(* PLC project paper-machine, Generated TextualNotationConverter 1.0 *)
(* stored: creationDateTime 2025-07-30T12:00:00, modificationDateTime 2025-01-30T12:00:00 *)

FUNCTION_BLOCK ANALOG_IN
  VAR_INPUT
    Name : STRING;
    Description : STRING;
    Raw_Signal : REAL;
    PV_High : REAL;
    PV_Low : REAL;
    Scaling_Slope : REAL;
    Scaling_Offset : REAL;
    Alarm_Enable : BOOL;
  END_VAR
  VAR_OUTPUT
    PV : REAL;
    High_Alarm : BOOL;
    Low_Alarm : BOOL;
    General_Fault : BOOL;
  END_VAR

            
          
END_FUNCTION_BLOCK

FUNCTION_BLOCK MOTOR_VSD
  VAR_INPUT
    Name : STRING;
    Description : STRING;
    Start_Cmd : BOOL;
    Stop_Cmd : BOOL;
    Speed_SP : REAL;
    Accel_Ramp : STRING;
    Decel_Ramp : STRING;
    Inhibit : BOOL;
  END_VAR
  VAR_OUTPUT
    Speed_Out : REAL;
    FB_Running : BOOL;
    FB_Fault : BOOL;
    FB_Ready : BOOL;
    FB_ActualSpeed : REAL;
    Alarm_Speed_Deviation : BOOL;
    Alarm_Comm_Fail : BOOL;
  END_VAR

            
          
END_FUNCTION_BLOCK

FUNCTION_BLOCK PID_BASIC
  VAR_INPUT
    Name : STRING;
    Description : STRING;
    AUTO : BOOL;
    PV : REAL;
    SP : REAL;
    MV_MIN : REAL;
    MV_MAX : REAL;
    X0 : REAL;
    KP : REAL;
    TR : REAL;
    TD : REAL;
    PV_High : REAL;
    PV_Low : REAL;
    Deviation_Limit : REAL;
    Inhibit : BOOL;
  END_VAR
  VAR_OUTPUT
    PV_High_Alarm : BOOL;
    PV_Low_Alarm : BOOL;
    Deviation_Alarm : BOOL;
    XOUT : REAL;
  END_VAR

            
          
END_FUNCTION_BLOCK

FUNCTION_BLOCK VALVE_ELECTRIC
  VAR_INPUT
    Name : STRING;
    Description : STRING;
    Control_Signal : REAL;
    Manual_Mode : BOOL;
    Manual_Position : REAL;
    Open_Limit : REAL;
    Close_Limit : REAL;
    Timeout : STRING;
    Inhibit : BOOL;
  END_VAR
  VAR_OUTPUT
    Valve_Position : REAL;
    Feedback_Pos : REAL;
    Valve_Moving : BOOL;
    Position_Error : BOOL;
    Alarm : BOOL;
  END_VAR

            
          
END_FUNCTION_BLOCK

FUNCTION_BLOCK VALVE_ON_OFF
  VAR_INPUT
    Name : STRING;
    Description : STRING;
    Open_Cmd : BOOL;
    Close_Cmd : BOOL;
    Timeout : STRING;
    Inhibit : BOOL;
  END_VAR
  VAR_OUTPUT
    FB_Opened : BOOL;
    FB_Closed : BOOL;
    Valve_Open_Out : BOOL;
    Valve_Close_Out : BOOL;
    Alarm_Position_Error : BOOL;
    Alarm_General : BOOL;
  END_VAR

            
          
END_FUNCTION_BLOCK

PROGRAM Section2
  VAR
    LT_101_Flow_PV : REAL;
    FC_101_MV_to_FV106 : REAL;
    M_102_VSD_Speed_Out : REAL;
    Flow_Deviation_Alarm_30s : BOOL;
    Flow_High_Alarm : BOOL;
    Flow_Low_Alarm : BOOL;
    M_102_Start_Request : BOOL;
    M_102_Stop_Request : BOOL;
  END_VAR
  VAR
    LT-101 : ANALOG_IN;
    FC-101 : PID_BASIC;
    M-102 : MOTOR_VSD;
    FV-106 : VALVE_ELECTRIC;
    LV-103 : VALVE_ELECTRIC;
    XV-102 : VALVE_ON_OFF;
    XV-104 : VALVE_ON_OFF;
    XV-105 : VALVE_ON_OFF;
  END_VAR
  VAR  (* added by the conversion: wires and edge detectors of the diagram *)
    _OR5_OUT : BOOL;
  END_VAR

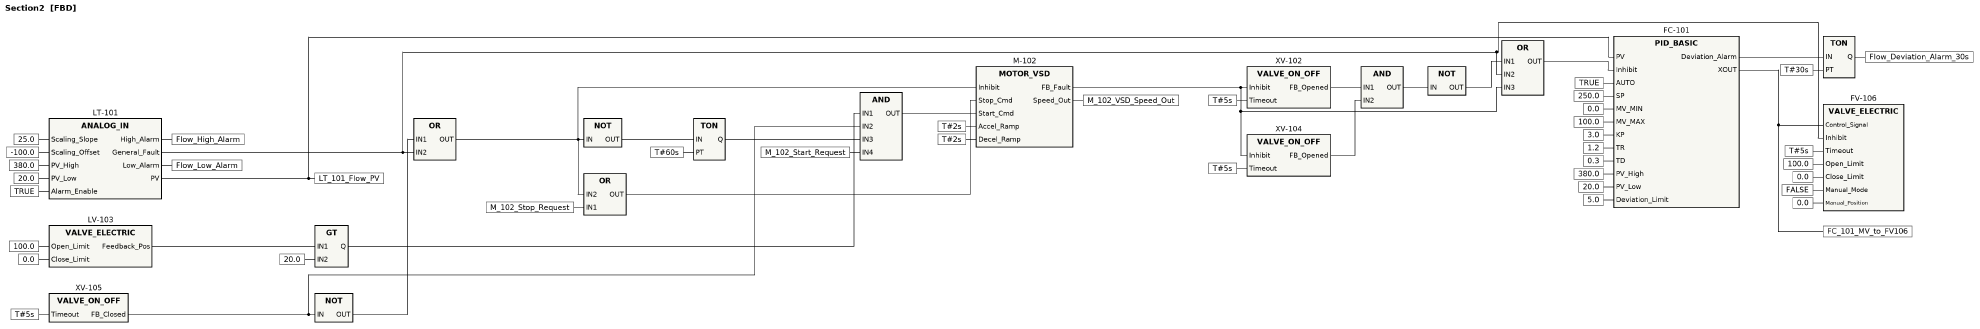
(* FBD diagram, written out as Structured Text *)
LT-101(Scaling_Slope := 25.0, Scaling_Offset := -100.0, PV_High := 380.0, PV_Low := 20.0, Alarm_Enable := TRUE);
XV-105(Timeout := T#5s);
_OR5_OUT := NOT XV-105.FB_Closed OR LT-101.General_Fault;
LV-103(Open_Limit := 100.0, Close_Limit := 0.0);
M-102(Inhibit := _OR5_OUT, Stop_Cmd := _OR5_OUT OR M_102_Stop_Request, Start_Cmd := LV-103.Feedback_Pos > 20.0 AND XV-105.FB_Closed AND TON(NOT _OR5_OUT, T#60s) AND M_102_Start_Request, Accel_Ramp := T#2s, Decel_Ramp := T#2s);
XV-102(Inhibit := M-102.FB_Fault, Timeout := T#5s);
XV-104(Inhibit := M-102.FB_Fault, Timeout := T#5s);
FC-101(PV := LT-101.PV, Inhibit := NOT (XV-102.FB_Opened AND XV-104.FB_Opened) OR LT-101.General_Fault OR M-102.FB_Fault, AUTO := TRUE, SP := 250.0, MV_MIN := 0.0, MV_MAX := 100.0, KP := 3.0, TR := 1.2, TD := 0.3, PV_High := 380.0, PV_Low := 20.0, Deviation_Limit := 5.0);
FC_101_MV_to_FV106 := FC-101.XOUT;
Flow_Deviation_Alarm_30s := TON(FC-101.Deviation_Alarm, T#30s);
Flow_High_Alarm := LT-101.High_Alarm;
Flow_Low_Alarm := LT-101.Low_Alarm;
LT_101_Flow_PV := LT-101.PV;
M_102_VSD_Speed_Out := M-102.Speed_Out;
FV-106(Control_Signal := FC-101.XOUT, Inhibit := LT-101.General_Fault, Timeout := T#5s, Open_Limit := 100.0, Close_Limit := 0.0, Manual_Mode := FALSE, Manual_Position := 0.0);
END_PROGRAM

FUNCTION_BLOCK BOOL_IN
  VAR_INPUT
    Name : STRING;
    Description : STRING;
    Bool_In : BOOL;
    Alarm_OnTrue : BOOL;
    Alarm_OnFalse : BOOL;
    Latch_Enable : BOOL;
    Reset_Latch : BOOL;
  END_VAR
  VAR_OUTPUT
    Bool_Out : BOOL;
    Alarm_Active : BOOL;
    Latched_Status : BOOL;
  END_VAR

            
          
END_FUNCTION_BLOCK

FUNCTION_BLOCK DIGITAL_IN
  VAR_INPUT
    Name : STRING;
    Description : STRING;
    DI_Raw : BOOL;
    DebounceTime : STRING;
    EnableAlarm : BOOL;
  END_VAR
  VAR_OUTPUT
    DI_Out : BOOL;
    Fault_State : BOOL;
  END_VAR

            
          
END_FUNCTION_BLOCK

FUNCTION_BLOCK DUTY_STANDBY
  VAR_INPUT
    Name : STRING;
    Description : STRING;
    Enable : BOOL;
    StartRequest : BOOL;
    AlternateEnable : BOOL;
    ForcePumpA : BOOL;
    ForcePumpB : BOOL;
    DutyElapsed : BOOL;
    MinRunElapsed : BOOL;
    SwitchoverDelayElapsed : BOOL;
    StartTimeoutElapsed : BOOL;
    PumpA_RunFB : BOOL;
    PumpB_RunFB : BOOL;
    PumpA_Fault : BOOL;
    PumpB_Fault : BOOL;
    Reset : BOOL;
    Inhibit : BOOL;
  END_VAR
  VAR_OUTPUT
    CmdPumpA : BOOL;
    CmdPumpB : BOOL;
    ActiveIsA : BOOL;
    SwitchedDueToDuty : BOOL;
    SwitchedDueToFailure : BOOL;
    Alarm_FailedStart_A : BOOL;
    Alarm_FailedStart_B : BOOL;
    Alarm_NoAvailablePump : BOOL;
  END_VAR

            
          
END_FUNCTION_BLOCK

FUNCTION_BLOCK MOTOR_2SPD
  VAR_INPUT
    Name : STRING;
    Description : STRING;
    Start_Cmd : BOOL;
    Stop_Cmd : BOOL;
    Speed_High_Cmd : BOOL;
    Speed_Low_Cmd : BOOL;
    Inhibit : BOOL;
  END_VAR
  VAR_OUTPUT
    Motor_Start_Out : BOOL;
    FB_Running : BOOL;
    FB_Trip : BOOL;
    FB_HighSpeed : BOOL;
    FB_LowSpeed : BOOL;
    Alarm_Speed_Error : BOOL;
  END_VAR

            
          
END_FUNCTION_BLOCK

FUNCTION_BLOCK MOTOR_ON_OFF
  VAR_INPUT
    Name : STRING;
    Description : STRING;
    Start_Cmd : BOOL;
    Stop_Cmd : BOOL;
    Start_Delay : STRING;
    MinRunTime : STRING;
    Inhibit : BOOL;
  END_VAR
  VAR_OUTPUT
    Motor_Start_Out : BOOL;
    FB_Running : BOOL;
    FB_Trip : BOOL;
    Alarm_Start_Fail : BOOL;
    Alarm_Stop_Fail : BOOL;
  END_VAR

            
          
END_FUNCTION_BLOCK

FUNCTION_BLOCK RATIO_CONTROL
  VAR_INPUT
    Name : STRING;
    Description : STRING;
    Auto : BOOL;
    PrimaryPV : REAL;
    SecondaryPV : REAL;
    RatioSP : REAL;
    Bias : REAL;
    TrimKp : REAL;
    TrimTi : STRING;
    MV_MIN : REAL;
    MV_MAX : REAL;
    ManOut : REAL;
    Inhibit : BOOL;
  END_VAR
  VAR_OUTPUT
    SlaveSP : REAL;
    ActiveRatio : REAL;
    RatioErr : REAL;
  END_VAR

            
          
END_FUNCTION_BLOCK

FUNCTION_BLOCK SPLIT_RANGE
  VAR_INPUT
    Name : STRING;
    Description : STRING;
    IN : REAL;
    Split_Point : REAL;
    Output1_Start : REAL;
    Output1_End : REAL;
    Output2_Start : REAL;
    Output2_End : REAL;
  END_VAR
  VAR_OUTPUT
    OUT1 : REAL;
    OUT2 : REAL;
  END_VAR

            
          
END_FUNCTION_BLOCK

FUNCTION_BLOCK VOTING_ANALOG
  VAR_INPUT
    Name : STRING;
    Description : STRING;
    Input1 : REAL;
    Input2 : REAL;
    Input3 : REAL;
    Deviation_Limit : REAL;
    Voting_Scheme : STRING;
    EnableAlarm : BOOL;
    Inhibit : BOOL;
  END_VAR
  VAR_OUTPUT
    Voted_Output : REAL;
    Sensor1_Fault : BOOL;
    Sensor2_Fault : BOOL;
    Sensor3_Fault : BOOL;
    Alarm_Voting_Error : BOOL;
    Healthy_Sensors_Count : INT;
  END_VAR

            
          
END_FUNCTION_BLOCK

PROGRAM Section3
  VAR
    TT_103_Temperature_PV : REAL;
    PT_101_Pressure_PV : REAL;
    TIC_104_RSP_to_FC_203 : REAL;
    PIC_101_RSP_to_FC_202 : REAL;
    FC_203_MV_to_SV_203 : REAL;
    FC_202_MV_to_FV_202 : REAL;
  END_VAR
  VAR
    TT-103 : ANALOG_IN;
    PT-101 : ANALOG_IN;
    TIC-104 : PID_BASIC;
    PIC-101 : PID_BASIC;
    FC-203 : PID_BASIC;
    FC-202 : PID_BASIC;
    SV-203 : VALVE_ELECTRIC;
    FV-202 : VALVE_ELECTRIC;
  END_VAR
  VAR  (* added by the conversion: wires and edge detectors of the diagram *)
    _OR59_OUT : BOOL;
  END_VAR

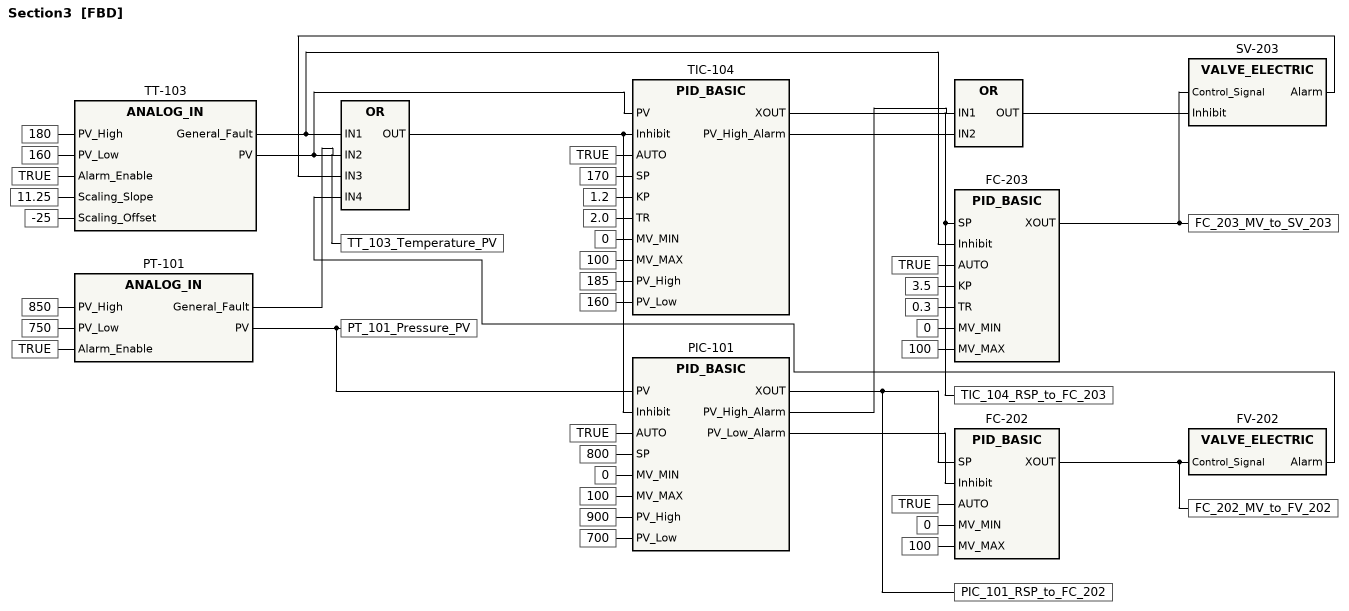
(* FBD diagram, written out as Structured Text *)
PT-101(PV_High := 850, PV_Low := 750, Alarm_Enable := TRUE);
TT-103(PV_High := 180, PV_Low := 160, Alarm_Enable := TRUE, Scaling_Slope := 11.25, Scaling_Offset := -25);
TIC-104(PV := TT-103.PV, Inhibit := _OR59_OUT, AUTO := TRUE, SP := 170, KP := 1.2, TR := 2.0, MV_MIN := 0, MV_MAX := 100, PV_High := 185, PV_Low := 160);
FC-203(SP := TIC-104.XOUT, Inhibit := TT-103.General_Fault, AUTO := TRUE, KP := 3.5, TR := 0.3, MV_MIN := 0, MV_MAX := 100);
SV-203(Control_Signal := FC-203.XOUT, Inhibit := PIC-101.PV_High_Alarm OR TIC-104.PV_High_Alarm);
FV-202(Control_Signal := FC-202.XOUT);
_OR59_OUT := TT-103.General_Fault OR PT-101.General_Fault OR SV-203.Alarm OR FV-202.Alarm;
PIC-101(PV := PT-101.PV, Inhibit := _OR59_OUT, AUTO := TRUE, SP := 800, MV_MIN := 0, MV_MAX := 100, PV_High := 900, PV_Low := 700);
FC-202(SP := PIC-101.XOUT, Inhibit := PIC-101.PV_Low_Alarm, AUTO := TRUE, MV_MIN := 0, MV_MAX := 100);
FC_202_MV_to_FV_202 := FC-202.XOUT;
FC_203_MV_to_SV_203 := FC-203.XOUT;
PIC_101_RSP_to_FC_202 := PIC-101.XOUT;
PT_101_Pressure_PV := PT-101.PV;
TIC_104_RSP_to_FC_203 := TIC-104.XOUT;
TT_103_Temperature_PV := TT-103.PV;
END_PROGRAM

PROGRAM Section4
  VAR
    PIT103_Pressure_kPa : REAL;
    PT101_UpstreamPressure_kPa : REAL;
    DT301_PulpDensity_Pct : REAL;
    PIC104_ControlOutput_to_FV106_Pct : REAL;
    FV106_ValvePositionFeedback_Pct : REAL;
  END_VAR
  VAR
    DT-301 : ANALOG_IN;
    PIT-103 : ANALOG_IN;
    PT-101 : ANALOG_IN;
    PIC-104 : PID_BASIC;
    FV-106 : VALVE_ELECTRIC;
    XV-102 : VALVE_ON_OFF;
    XV-107 : VALVE_ON_OFF;
    XV-102-OPEN-FB : DIGITAL_IN;
    XV-107-OPEN-FB : DIGITAL_IN;
    PERM-XV102-OPEN : BOOL_IN;
    PERM-XV107-OPEN : BOOL_IN;
  END_VAR
  VAR  (* added by the conversion: wires and edge detectors of the diagram *)
    _OR104_OUT : BOOL;
    _OR106_OUT : BOOL;
    _NOT109_OUT : BOOL;
  END_VAR

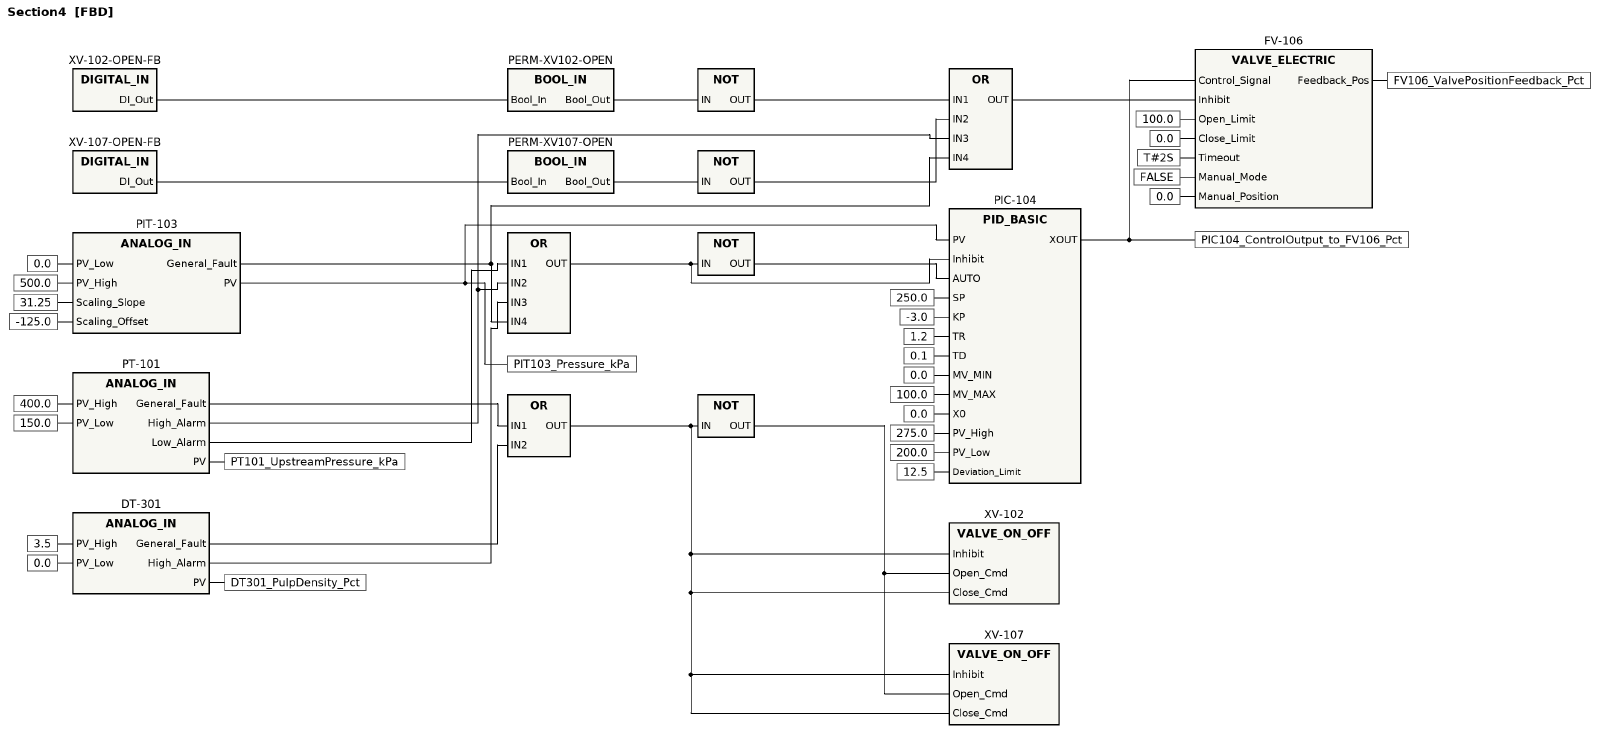
(* FBD diagram, written out as Structured Text *)
DT-301(PV_High := 3.5, PV_Low := 0.0);
DT301_PulpDensity_Pct := DT-301.PV;
PIT-103(PV_Low := 0.0, PV_High := 500.0, Scaling_Slope := 31.25, Scaling_Offset := -125.0);
PT-101(PV_High := 400.0, PV_Low := 150.0);
_OR104_OUT := PT-101.Low_Alarm OR PT-101.High_Alarm OR DT-301.High_Alarm OR PIT-103.General_Fault;
PIC-104(PV := PIT-103.PV, Inhibit := _OR104_OUT, AUTO := NOT _OR104_OUT, SP := 250.0, KP := -3.0, TR := 1.2, TD := 0.1, MV_MIN := 0.0, MV_MAX := 100.0, X0 := 0.0, PV_High := 275.0, PV_Low := 200.0, Deviation_Limit := 12.5);
XV-102-OPEN-FB();
PERM-XV102-OPEN(Bool_In := XV-102-OPEN-FB.DI_Out);
XV-107-OPEN-FB();
PERM-XV107-OPEN(Bool_In := XV-107-OPEN-FB.DI_Out);
FV-106(Control_Signal := PIC-104.XOUT, Inhibit := NOT PERM-XV102-OPEN.Bool_Out OR NOT PERM-XV107-OPEN.Bool_Out OR PT-101.High_Alarm OR PIT-103.General_Fault, Open_Limit := 100.0, Close_Limit := 0.0, Timeout := T#2S, Manual_Mode := FALSE, Manual_Position := 0.0);
FV106_ValvePositionFeedback_Pct := FV-106.Feedback_Pos;
PIC104_ControlOutput_to_FV106_Pct := PIC-104.XOUT;
PIT103_Pressure_kPa := PIT-103.PV;
PT101_UpstreamPressure_kPa := PT-101.PV;
_OR106_OUT := PT-101.General_Fault OR DT-301.General_Fault;
_NOT109_OUT := NOT _OR106_OUT;
XV-102(Inhibit := _OR106_OUT, Open_Cmd := _NOT109_OUT, Close_Cmd := _OR106_OUT);
XV-107(Inhibit := _OR106_OUT, Open_Cmd := _NOT109_OUT, Close_Cmd := _OR106_OUT);
END_PROGRAM

PROGRAM Section5
  VAR
    AT102_pH_PV : REAL;
    AT107_pH_PV : REAL;
    TIT106_Temperature_PV : REAL;
    LIC102_MV_to_FV101 : REAL;
    TIC106_MV_to_FV103 : REAL;
    LIC104_MV_to_XV104 : REAL;
  END_VAR
  VAR
    AT-102 : ANALOG_IN;
    AT-107 : ANALOG_IN;
    TIT-106 : ANALOG_IN;
    LIC-102 : PID_BASIC;
    TIC-106 : PID_BASIC;
    LIC-104 : PID_BASIC;
    FV-101 : VALVE_ELECTRIC;
    FV-103 : VALVE_ELECTRIC;
    XV-104 : VALVE_ELECTRIC;
  END_VAR

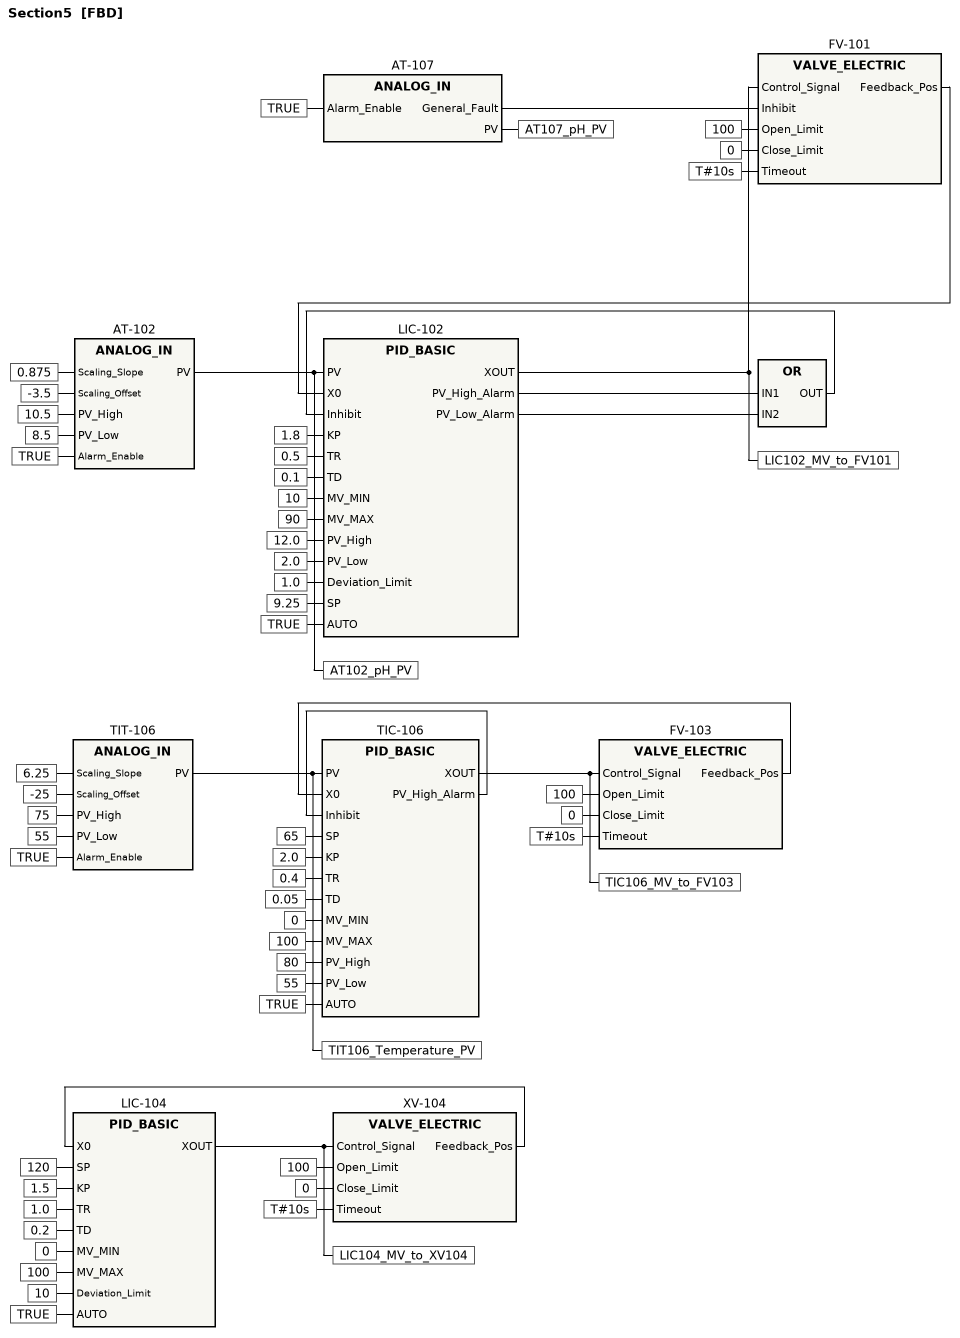
(* FBD diagram, written out as Structured Text *)
AT-102(Scaling_Slope := 0.875, Scaling_Offset := -3.5, PV_High := 10.5, PV_Low := 8.5, Alarm_Enable := TRUE);
AT102_pH_PV := AT-102.PV;
AT-107(Alarm_Enable := TRUE);
AT107_pH_PV := AT-107.PV;
FV-101(Control_Signal := LIC-102.XOUT, Inhibit := AT-107.General_Fault, Open_Limit := 100, Close_Limit := 0, Timeout := T#10s);
LIC-102(PV := AT-102.PV, X0 := FV-101.Feedback_Pos, Inhibit := LIC-102.PV_High_Alarm OR LIC-102.PV_Low_Alarm, KP := 1.8, TR := 0.5, TD := 0.1, MV_MIN := 10, MV_MAX := 90, PV_High := 12.0, PV_Low := 2.0, Deviation_Limit := 1.0, SP := 9.25, AUTO := TRUE);
LIC102_MV_to_FV101 := LIC-102.XOUT;
XV-104(Control_Signal := LIC-104.XOUT, Open_Limit := 100, Close_Limit := 0, Timeout := T#10s);
LIC-104(X0 := XV-104.Feedback_Pos, SP := 120, KP := 1.5, TR := 1.0, TD := 0.2, MV_MIN := 0, MV_MAX := 100, Deviation_Limit := 10, AUTO := TRUE);
LIC104_MV_to_XV104 := LIC-104.XOUT;
TIT-106(Scaling_Slope := 6.25, Scaling_Offset := -25, PV_High := 75, PV_Low := 55, Alarm_Enable := TRUE);
FV-103(Control_Signal := TIC-106.XOUT, Open_Limit := 100, Close_Limit := 0, Timeout := T#10s);
TIC-106(PV := TIT-106.PV, X0 := FV-103.Feedback_Pos, Inhibit := TIC-106.PV_High_Alarm, SP := 65, KP := 2.0, TR := 0.4, TD := 0.05, MV_MIN := 0, MV_MAX := 100, PV_High := 80, PV_Low := 55, AUTO := TRUE);
TIC106_MV_to_FV103 := TIC-106.XOUT;
TIT106_Temperature_PV := TIT-106.PV;
END_PROGRAM

PROGRAM Section6
  VAR
    CT501_Consistency_PV_Pct : REAL;
    FC502_MV_to_FV502_Pct : REAL;
    SELT501_SEL_PV_WsPerMm2 : REAL;
    SELC501_MV_to_PGA501_Pct : REAL;
    LT501_Level_PV_Pct : REAL;
    PT502_Pressure_PV_kPa : REAL;
    PGT501_PlateGap_PV_mm : REAL;
  END_VAR
  VAR
    CT-501 : ANALOG_IN;
    FC-502 : PID_BASIC;
    FV-502 : VALVE_ELECTRIC;
    LT-501 : ANALOG_IN;
    M-501 : MOTOR_ON_OFF;
    PT-502 : ANALOG_IN;
    SELC-501 : PID_BASIC;
    PGT-501 : ANALOG_IN;
    PGA-501 : VALVE_ELECTRIC;
    SELT-501 : ANALOG_IN;
    INTLK-M501-RUNNING : BOOL_IN;
    INTLK-PLATE-GAP-IN-RANGE : BOOL_IN;
    INTLK-LEVEL-ABOVE-20 : BOOL_IN;
    PERM-PT502-IN-RANGE : BOOL_IN;
  END_VAR
  VAR  (* added by the conversion: wires and edge detectors of the diagram *)
    _OR217_OUT : BOOL;
    _OR219_OUT : BOOL;
    _OR221_OUT : BOOL;
    _OR213_OUT : BOOL;
  END_VAR

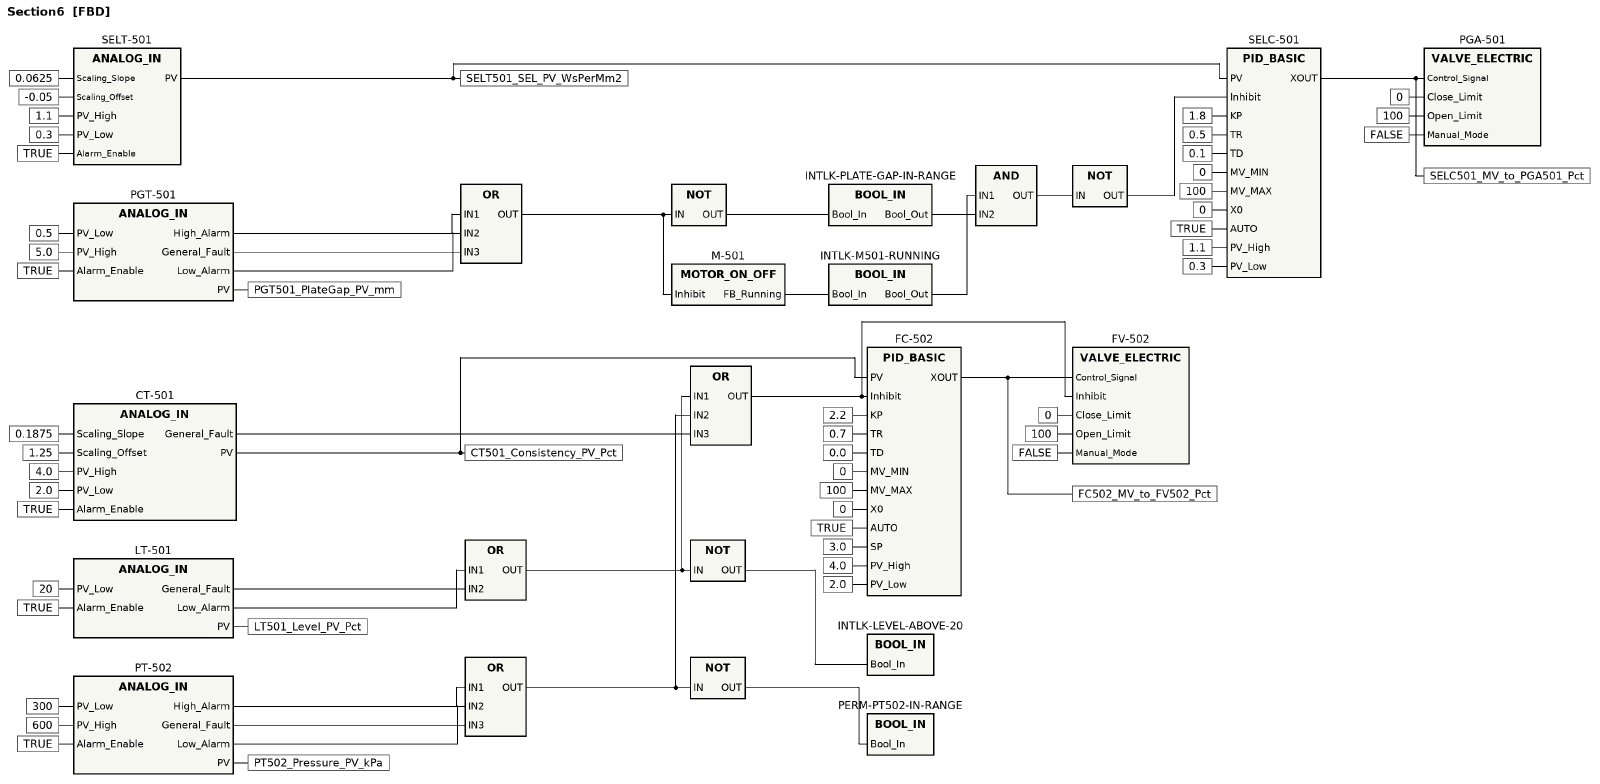
(* FBD diagram, written out as Structured Text *)
CT-501(Scaling_Slope := 0.1875, Scaling_Offset := 1.25, PV_High := 4.0, PV_Low := 2.0, Alarm_Enable := TRUE);
CT501_Consistency_PV_Pct := CT-501.PV;
LT-501(PV_Low := 20, Alarm_Enable := TRUE);
_OR217_OUT := LT-501.Low_Alarm OR LT-501.General_Fault;
PT-502(PV_Low := 300, PV_High := 600, Alarm_Enable := TRUE);
_OR219_OUT := PT-502.High_Alarm OR PT-502.Low_Alarm OR PT-502.General_Fault;
_OR221_OUT := _OR217_OUT OR _OR219_OUT OR CT-501.General_Fault;
FC-502(PV := CT-501.PV, Inhibit := _OR221_OUT, KP := 2.2, TR := 0.7, TD := 0.0, MV_MIN := 0, MV_MAX := 100, X0 := 0, AUTO := TRUE, SP := 3.0, PV_High := 4.0, PV_Low := 2.0);
FC502_MV_to_FV502_Pct := FC-502.XOUT;
LT501_Level_PV_Pct := LT-501.PV;
PGT-501(PV_Low := 0.5, PV_High := 5.0, Alarm_Enable := TRUE);
PGT501_PlateGap_PV_mm := PGT-501.PV;
PT502_Pressure_PV_kPa := PT-502.PV;
SELT-501(Scaling_Slope := 0.0625, Scaling_Offset := -0.05, PV_High := 1.1, PV_Low := 0.3, Alarm_Enable := TRUE);
_OR213_OUT := PGT-501.High_Alarm OR PGT-501.Low_Alarm OR PGT-501.General_Fault;
M-501(Inhibit := _OR213_OUT);
INTLK-M501-RUNNING(Bool_In := M-501.FB_Running);
INTLK-PLATE-GAP-IN-RANGE(Bool_In := NOT _OR213_OUT);
SELC-501(PV := SELT-501.PV, Inhibit := NOT (INTLK-M501-RUNNING.Bool_Out AND INTLK-PLATE-GAP-IN-RANGE.Bool_Out), KP := 1.8, TR := 0.5, TD := 0.1, MV_MIN := 0, MV_MAX := 100, X0 := 0, AUTO := TRUE, PV_High := 1.1, PV_Low := 0.3);
SELC501_MV_to_PGA501_Pct := SELC-501.XOUT;
SELT501_SEL_PV_WsPerMm2 := SELT-501.PV;
FV-502(Control_Signal := FC-502.XOUT, Inhibit := _OR221_OUT, Close_Limit := 0, Open_Limit := 100, Manual_Mode := FALSE);
PGA-501(Control_Signal := SELC-501.XOUT, Close_Limit := 0, Open_Limit := 100, Manual_Mode := FALSE);
INTLK-LEVEL-ABOVE-20(Bool_In := NOT _OR217_OUT);
PERM-PT502-IN-RANGE(Bool_In := NOT _OR219_OUT);
END_PROGRAM

PROGRAM Section7
  VAR
    CT_601_PV : REAL;
    FT_601_PV : REAL;
    FT_601_SP : REAL;
    PIT_601_PV : REAL;
    VT_601_PV : REAL;
    FS_601_MinFlow_OK : BOOL;
    P_601_Run_OK : BOOL;
    FFIC601_Bias : REAL;
    ALM_601 : BOOL;
    ALM_601_High : BOOL;
    ALM_601_Low : BOOL;
    ALM_602 : BOOL;
    ALM_603 : BOOL;
    ALM_604 : BOOL;
    Process_Permissives_OK : BOOL;
    MasterInhibit : BOOL;
    CT601_RateHigh : BOOL;
  END_VAR
  VAR
    CT-601 : ANALOG_IN;
    FT-601 : ANALOG_IN;
    PIT-601 : ANALOG_IN;
    VT-601 : ANALOG_IN;
    FS-601 : BOOL_IN;
    P-601_RUN : BOOL_IN;
    FV-601 : VALVE_ELECTRIC;
    FIC-601 : PID_BASIC;
    FFIC-601 : RATIO_CONTROL;
    ProcessUpset_Timer : TON;
  END_VAR
  VAR  (* added by the conversion: wires and edge detectors of the diagram *)
    _OR288_OUT : BOOL;
    _OR289_OUT : BOOL;
    _OR290_OUT : BOOL;
    _NOT291_OUT : BOOL;
  END_VAR

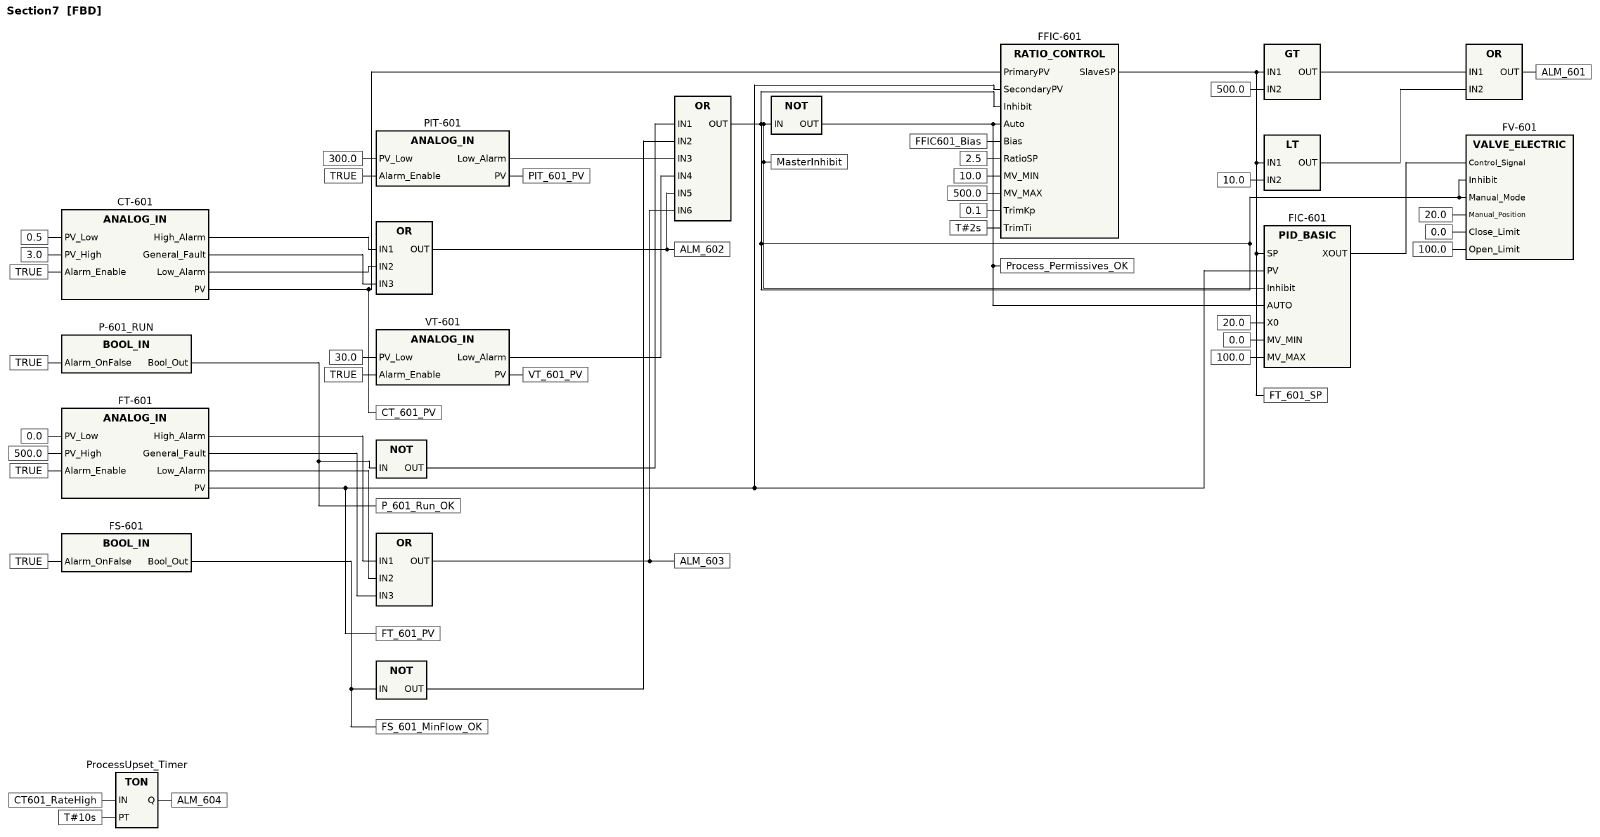
(* FBD diagram, written out as Structured Text *)
CT-601(PV_Low := 0.5, PV_High := 3.0, Alarm_Enable := TRUE);
FT-601(PV_Low := 0.0, PV_High := 500.0, Alarm_Enable := TRUE);
P-601_RUN(Alarm_OnFalse := TRUE);
FS-601(Alarm_OnFalse := TRUE);
PIT-601(PV_Low := 300.0, Alarm_Enable := TRUE);
VT-601(PV_Low := 30.0, Alarm_Enable := TRUE);
_OR288_OUT := CT-601.High_Alarm OR CT-601.Low_Alarm OR CT-601.General_Fault;
_OR289_OUT := FT-601.High_Alarm OR FT-601.Low_Alarm OR FT-601.General_Fault;
_OR290_OUT := NOT P-601_RUN.Bool_Out OR NOT FS-601.Bool_Out OR PIT-601.Low_Alarm OR VT-601.Low_Alarm OR _OR288_OUT OR _OR289_OUT;
_NOT291_OUT := NOT _OR290_OUT;
FFIC-601(PrimaryPV := CT-601.PV, SecondaryPV := FT-601.PV, Inhibit := _OR290_OUT, Auto := _NOT291_OUT, Bias := FFIC601_Bias, RatioSP := 2.5, MV_MIN := 10.0, MV_MAX := 500.0, TrimKp := 0.1, TrimTi := T#2s);
ALM_601 := FFIC-601.SlaveSP > 500.0 OR FFIC-601.SlaveSP < 10.0;
ALM_602 := _OR288_OUT;
ALM_603 := _OR289_OUT;
ProcessUpset_Timer(IN := CT601_RateHigh, PT := T#10s);
ALM_604 := ProcessUpset_Timer.Q;
CT_601_PV := CT-601.PV;
FS_601_MinFlow_OK := FS-601.Bool_Out;
FT_601_PV := FT-601.PV;
FT_601_SP := FFIC-601.SlaveSP;
MasterInhibit := _OR290_OUT;
PIT_601_PV := PIT-601.PV;
P_601_Run_OK := P-601_RUN.Bool_Out;
Process_Permissives_OK := _NOT291_OUT;
VT_601_PV := VT-601.PV;
FIC-601(SP := FFIC-601.SlaveSP, PV := FT-601.PV, Inhibit := _OR290_OUT, AUTO := _NOT291_OUT, X0 := 20.0, MV_MIN := 0.0, MV_MAX := 100.0);
FV-601(Control_Signal := FIC-601.XOUT, Inhibit := _OR290_OUT, Manual_Mode := _OR290_OUT, Manual_Position := 20.0, Close_Limit := 0.0, Open_Limit := 100.0);
END_PROGRAM

PROGRAM Section8
  VAR
    MM701_Raw_mA : REAL;
    PT701_Raw : REAL;
    TT102_Raw : REAL;
    HS701_ON : BOOL;
    CS701_ON : BOOL;
    SB701_SheetBreak : BOOL;
    MM701_Moisture_PV : REAL;
    PT701_HydraulicPressure_PV : REAL;
    TT102_ShowerWaterTemp_PV : REAL;
    PV101_Pressure_Command_Pct : REAL;
    PV101_Position_Feedback_Pct : REAL;
    ESD_Trip : BOOL;
  END_VAR
  VAR
    MM-701 : ANALOG_IN;
    PT-701 : ANALOG_IN;
    TT-102 : ANALOG_IN;
    LIC-701 : PID_BASIC;
    PV-101 : VALVE_ELECTRIC;
    HS-701 : BOOL_IN;
    CS-701 : BOOL_IN;
    SB-701 : BOOL_IN;
  END_VAR
  VAR  (* added by the conversion: wires and edge detectors of the diagram *)
    _OR348_OUT : BOOL;
  END_VAR

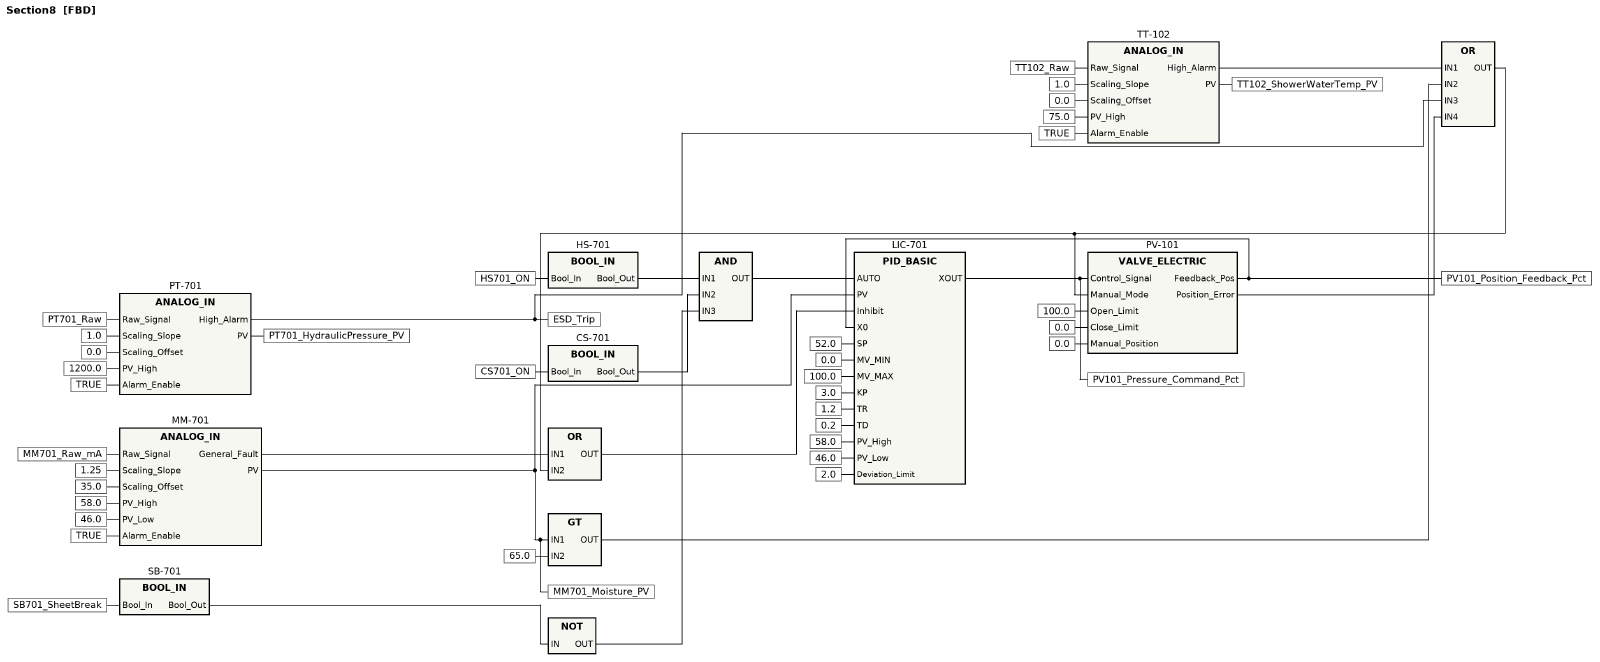
(* FBD diagram, written out as Structured Text *)
PT-701(Raw_Signal := PT701_Raw, Scaling_Slope := 1.0, Scaling_Offset := 0.0, PV_High := 1200.0, Alarm_Enable := TRUE);
ESD_Trip := PT-701.High_Alarm;
MM-701(Raw_Signal := MM701_Raw_mA, Scaling_Slope := 1.25, Scaling_Offset := 35.0, PV_High := 58.0, PV_Low := 46.0, Alarm_Enable := TRUE);
MM701_Moisture_PV := MM-701.PV;
PT701_HydraulicPressure_PV := PT-701.PV;
HS-701(Bool_In := HS701_ON);
CS-701(Bool_In := CS701_ON);
SB-701(Bool_In := SB701_SheetBreak);
TT-102(Raw_Signal := TT102_Raw, Scaling_Slope := 1.0, Scaling_Offset := 0.0, PV_High := 75.0, Alarm_Enable := TRUE);
_OR348_OUT := TT-102.High_Alarm OR MM-701.PV > 65.0 OR PT-701.High_Alarm OR PV-101.Position_Error;
LIC-701(AUTO := HS-701.Bool_Out AND CS-701.Bool_Out AND NOT SB-701.Bool_Out, PV := MM-701.PV, Inhibit := MM-701.General_Fault OR _OR348_OUT, X0 := PV-101.Feedback_Pos, SP := 52.0, MV_MIN := 0.0, MV_MAX := 100.0, KP := 3.0, TR := 1.2, TD := 0.2, PV_High := 58.0, PV_Low := 46.0, Deviation_Limit := 2.0);
PV-101(Control_Signal := LIC-701.XOUT, Manual_Mode := _OR348_OUT, Open_Limit := 100.0, Close_Limit := 0.0, Manual_Position := 0.0);
PV101_Position_Feedback_Pct := PV-101.Feedback_Pos;
PV101_Pressure_Command_Pct := LIC-701.XOUT;
TT102_ShowerWaterTemp_PV := TT-102.PV;
END_PROGRAM

PROGRAM Section9
  VAR
    F801_ExhaustFan_Speed_CMD_PCT : REAL;
    FV801_SteamFlowValve_Position_CMD_PCT : REAL;
    XV802_HotAirDamper_Position_CMD_PCT : REAL;
    WT801_DownstreamDriveRoll_Torque_CMD_PCT : REAL;
    XV802_Open_FB : BOOL;
    IR801_Available : BOOL;
  END_VAR
  VAR
    TT-801 : ANALOG_IN;
    TT-802 : ANALOG_IN;
    PT-801 : ANALOG_IN;
    IR-801 : ANALOG_IN;
    WT-801 : ANALOG_IN;
    F-801 : MOTOR_VSD;
    M-801 : MOTOR_ON_OFF;
    FV-801 : VALVE_ELECTRIC;
    XV-802 : VALVE_ELECTRIC;
    SC-801 : PID_BASIC;
    TC-801 : PID_BASIC;
    F-801_CTRL : PID_BASIC;
    WT-801_CTRL : PID_BASIC;
  END_VAR
  VAR  (* added by the conversion: wires and edge detectors of the diagram *)
    _OR401_OUT : BOOL;
    _OR397_OUT : BOOL;
  END_VAR

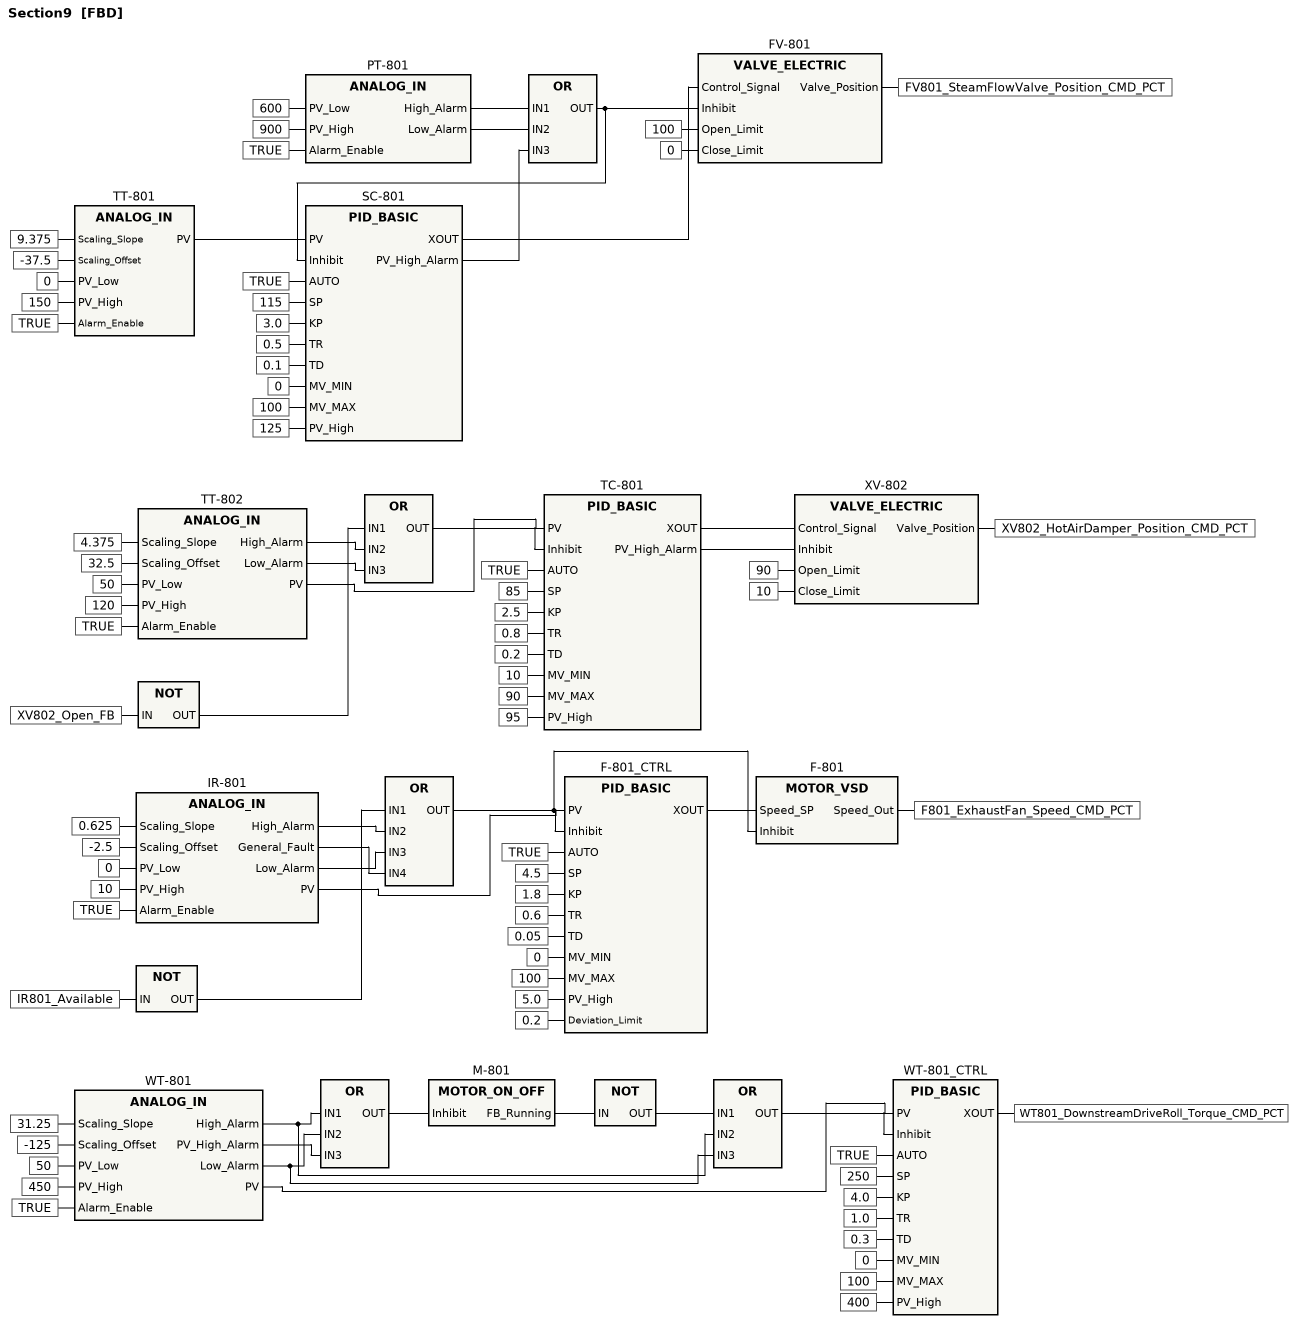
(* FBD diagram, written out as Structured Text *)
IR-801(Scaling_Slope := 0.625, Scaling_Offset := -2.5, PV_Low := 0, PV_High := 10, Alarm_Enable := TRUE);
_OR401_OUT := NOT IR801_Available OR IR-801.High_Alarm OR IR-801.Low_Alarm OR IR-801.General_Fault;
F-801_CTRL(PV := IR-801.PV, Inhibit := _OR401_OUT, AUTO := TRUE, SP := 4.5, KP := 1.8, TR := 0.6, TD := 0.05, MV_MIN := 0, MV_MAX := 100, PV_High := 5.0, Deviation_Limit := 0.2);
F-801(Speed_SP := F-801_CTRL.XOUT, Inhibit := _OR401_OUT);
F801_ExhaustFan_Speed_CMD_PCT := F-801.Speed_Out;
TT-801(Scaling_Slope := 9.375, Scaling_Offset := -37.5, PV_Low := 0, PV_High := 150, Alarm_Enable := TRUE);
PT-801(PV_Low := 600, PV_High := 900, Alarm_Enable := TRUE);
_OR397_OUT := PT-801.High_Alarm OR PT-801.Low_Alarm OR SC-801.PV_High_Alarm;
SC-801(PV := TT-801.PV, Inhibit := _OR397_OUT, AUTO := TRUE, SP := 115, KP := 3.0, TR := 0.5, TD := 0.1, MV_MIN := 0, MV_MAX := 100, PV_High := 125);
FV-801(Control_Signal := SC-801.XOUT, Inhibit := _OR397_OUT, Open_Limit := 100, Close_Limit := 0);
FV801_SteamFlowValve_Position_CMD_PCT := FV-801.Valve_Position;
WT-801(Scaling_Slope := 31.25, Scaling_Offset := -125, PV_Low := 50, PV_High := 450, Alarm_Enable := TRUE);
M-801(Inhibit := WT-801.High_Alarm OR WT-801.Low_Alarm OR WT-801.PV_High_Alarm);
WT-801_CTRL(PV := WT-801.PV, Inhibit := NOT M-801.FB_Running OR WT-801.High_Alarm OR WT-801.Low_Alarm, AUTO := TRUE, SP := 250, KP := 4.0, TR := 1.0, TD := 0.3, MV_MIN := 0, MV_MAX := 100, PV_High := 400);
WT801_DownstreamDriveRoll_Torque_CMD_PCT := WT-801_CTRL.XOUT;
TT-802(Scaling_Slope := 4.375, Scaling_Offset := 32.5, PV_Low := 50, PV_High := 120, Alarm_Enable := TRUE);
TC-801(PV := TT-802.PV, Inhibit := NOT XV802_Open_FB OR TT-802.High_Alarm OR TT-802.Low_Alarm, AUTO := TRUE, SP := 85, KP := 2.5, TR := 0.8, TD := 0.2, MV_MIN := 10, MV_MAX := 90, PV_High := 95);
XV-802(Control_Signal := TC-801.XOUT, Inhibit := TC-801.PV_High_Alarm, Open_Limit := 90, Close_Limit := 10);
XV802_HotAirDamper_Position_CMD_PCT := XV-802.Valve_Position;
END_PROGRAM

PROGRAM Section10
  VAR
    FT901_NipLoad_kN : REAL;
    FT902_FlowRate_Lmin : REAL;
    FIC904_Flow_SP_FromRatio : REAL;
  END_VAR
  VAR
    FT-901 : ANALOG_IN;
    FT-902 : ANALOG_IN;
    CW-901 : ANALOG_IN;
    FFIC-903 : RATIO_CONTROL;
    FIC-904 : PID_BASIC;
    FV-104 : VALVE_ELECTRIC;
    XV-105 : VALVE_ON_OFF;
  END_VAR
  VAR  (* added by the conversion: wires and edge detectors of the diagram *)
    _OR492_OUT : BOOL;
  END_VAR

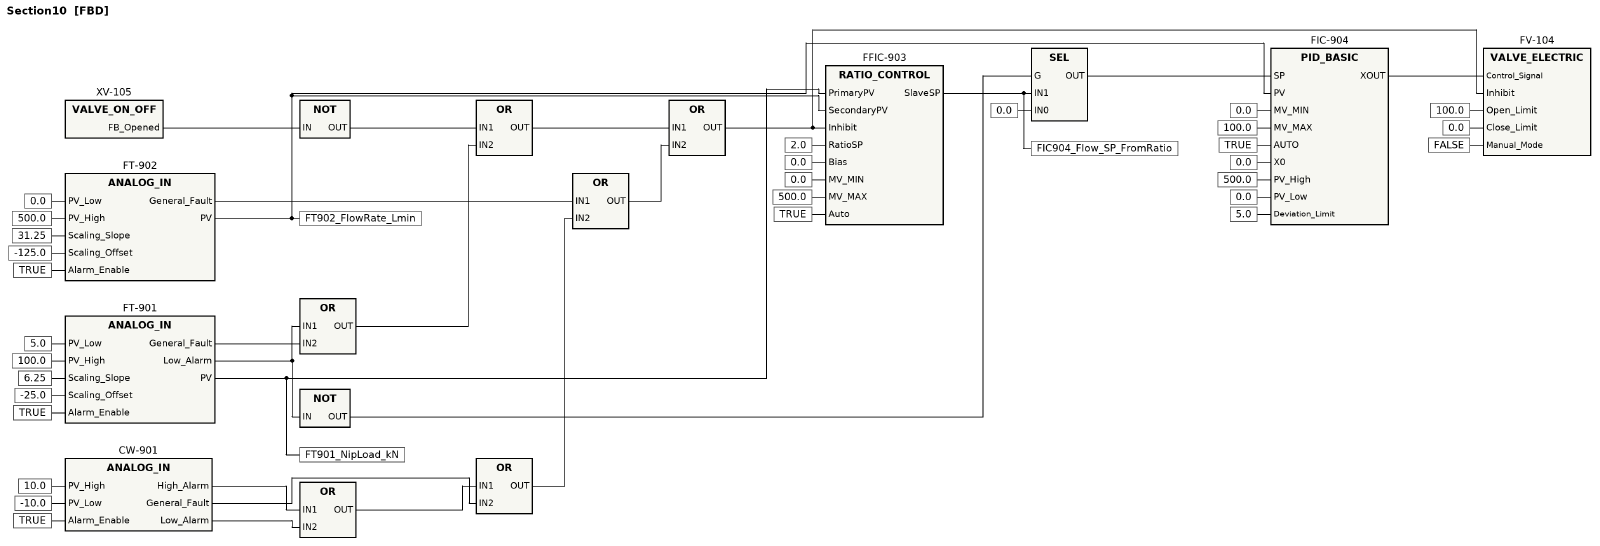
(* FBD diagram, written out as Structured Text *)
FT-901(PV_Low := 5.0, PV_High := 100.0, Scaling_Slope := 6.25, Scaling_Offset := -25.0, Alarm_Enable := TRUE);
FT-902(PV_Low := 0.0, PV_High := 500.0, Scaling_Slope := 31.25, Scaling_Offset := -125.0, Alarm_Enable := TRUE);
XV-105();
CW-901(PV_High := 10.0, PV_Low := -10.0, Alarm_Enable := TRUE);
_OR492_OUT := NOT XV-105.FB_Opened OR FT-901.Low_Alarm OR FT-901.General_Fault OR FT-902.General_Fault OR CW-901.High_Alarm OR CW-901.Low_Alarm OR CW-901.General_Fault;
FFIC-903(PrimaryPV := FT-901.PV, SecondaryPV := FT-902.PV, Inhibit := _OR492_OUT, RatioSP := 2.0, Bias := 0.0, MV_MIN := 0.0, MV_MAX := 500.0, Auto := TRUE);
FIC904_Flow_SP_FromRatio := FFIC-903.SlaveSP;
FT901_NipLoad_kN := FT-901.PV;
FT902_FlowRate_Lmin := FT-902.PV;
FIC-904(SP := SEL(NOT FT-901.Low_Alarm, FFIC-903.SlaveSP, 0.0), PV := FT-902.PV, MV_MIN := 0.0, MV_MAX := 100.0, AUTO := TRUE, X0 := 0.0, PV_High := 500.0, PV_Low := 0.0, Deviation_Limit := 5.0);
FV-104(Control_Signal := FIC-904.XOUT, Inhibit := _OR492_OUT, Open_Limit := 100.0, Close_Limit := 0.0, Manual_Mode := FALSE);
END_PROGRAM

CONFIGURATION Config0
  RESOURCE Res0 ON PLC
    TASK task0(INTERVAL := T#20ms, PRIORITY := 0);
    PROGRAM instance0 WITH task0 : Section2;
    PROGRAM instance_1 WITH task0 : Section3;
    PROGRAM instance_2 WITH task0 : Section4;
    PROGRAM instance_3 WITH task0 : Section5;
    PROGRAM instance_4 WITH task0 : Section6;
    PROGRAM instance_5 WITH task0 : Section7;
    PROGRAM instance_6 WITH task0 : Section8;
    PROGRAM instance_7 WITH task0 : Section9;
    PROGRAM instance_8 WITH task0 : Section10;
  END_RESOURCE
END_CONFIGURATION
